DATA_BLOCK "CS_Drive_TL"   // DB14, Motion_DB
// stored: InstanceOfName TO_SynchronousAxis, OfSystemLibElement TO_SynchronousAxis, OfSystemLibVersion 7.0
TO_SynchronousAxis   // technology object, version 7.0
// stored: Connection Interface Actor, InputAddress 816, OutputAddress 816
// stored: Connection Interface Sensor[1], InputAddress 816, OutputAddress 816, SensorIndexInActorTelegram 1
   // // inherited from TO_PositioningAxis
   // // inherited from TO_SpeedAxis
   // // inherited from TO_Axis
   // // inherited from TO_Object
   // VAR
   //    Actor : TO_Struct_Actor;
   // END_VAR
   // VAR
   //    Sensor : Array[1..4] of TO_Struct_Sensor;
   //    PositionControl : TO_Struct_PositionControl;
   // END_VAR
   // VAR
   //    StatusSynchronizedMotion { ExternalWritable := 'False'; S7_SetPoint := 'True'} : TO_Struct_StatusSynchronizedMotion;
   // END_VAR
BEGIN
   Actor.Interface.AddressIn.RID := 16#208072a;
   Actor.Interface.AddressIn.AREA := 16#81;
   Actor.Interface.AddressIn.OFFSET := 816;
   Actor.Interface.AddressOut.RID := 16#208072b;
   Actor.Interface.AddressOut.AREA := 16#82;
   Actor.Interface.AddressOut.OFFSET := 816;
   Sensor[1].Interface.AddressIn.RID := 16#208072a;
   Sensor[1].Interface.AddressIn.AREA := 16#81;
   Sensor[1].Interface.AddressIn.OFFSET := 816;
   Sensor[1].Interface.AddressOut.RID := 16#208072b;
   Sensor[1].Interface.AddressOut.AREA := 16#82;
   Sensor[1].Interface.AddressOut.OFFSET := 816;
   PositionControl.EnableDSC := true;
   _Actor.Interface.Telegram := 105;
   _Sensor[1].Interface.Telegram := 105;
END_DATA_BLOCK

DATA_BLOCK "CS_Drive_TP"   // DB13, Motion_DB
// stored: InstanceOfName TO_SynchronousAxis, OfSystemLibElement TO_SynchronousAxis, OfSystemLibVersion 7.0
TO_SynchronousAxis   // technology object, version 7.0
// stored: Connection Interface Actor, InputAddress 608, OutputAddress 608
// stored: Connection Interface Sensor[1], InputAddress 608, OutputAddress 608, SensorIndexInActorTelegram 1
   // // inherited from TO_PositioningAxis
   // // inherited from TO_SpeedAxis
   // // inherited from TO_Axis
   // // inherited from TO_Object
   // VAR
   //    Actor : TO_Struct_Actor;
   // END_VAR
   // VAR
   //    Sensor : Array[1..4] of TO_Struct_Sensor;
   //    PositionControl : TO_Struct_PositionControl;
   // END_VAR
   // VAR
   //    StatusSynchronizedMotion { ExternalWritable := 'False'; S7_SetPoint := 'True'} : TO_Struct_StatusSynchronizedMotion;
   // END_VAR
BEGIN
   Actor.Interface.AddressIn.RID := 16#208072a;
   Actor.Interface.AddressIn.AREA := 16#81;
   Actor.Interface.AddressIn.OFFSET := 608;
   Actor.Interface.AddressOut.RID := 16#208072b;
   Actor.Interface.AddressOut.AREA := 16#82;
   Actor.Interface.AddressOut.OFFSET := 608;
   Sensor[1].Interface.AddressIn.RID := 16#208072a;
   Sensor[1].Interface.AddressIn.AREA := 16#81;
   Sensor[1].Interface.AddressIn.OFFSET := 608;
   Sensor[1].Interface.AddressOut.RID := 16#208072b;
   Sensor[1].Interface.AddressOut.AREA := 16#82;
   Sensor[1].Interface.AddressOut.OFFSET := 608;
   PositionControl.EnableDSC := true;
   _Actor.Interface.Telegram := 105;
   _Sensor[1].Interface.Telegram := 105;
END_DATA_BLOCK

DATA_BLOCK "CS_Virtual_Axis"   // DB22, Motion_DB
// stored: InstanceOfName TO_PositioningAxis, OfSystemLibElement TO_PositioningAxis, OfSystemLibVersion 7.0
TO_PositioningAxis   // technology object, version 7.0
   // // inherited from TO_SpeedAxis
   // // inherited from TO_Axis
   // // inherited from TO_Object
   // VAR
   //    VirtualAxis : TO_Struct_VirtualAxis;
   // END_VAR
   // VAR
   //    Position { ExternalWritable := 'False'} : LReal;
   //    ActualPosition { ExternalWritable := 'False'} : LReal;
   //    ActualVelocity { ExternalWritable := 'False'} : LReal;
   //    ActualAcceleration { ExternalWritable := 'False'} : LReal;
   //    OperativeSensor { ExternalWritable := 'False'} : UDInt;
   //    ModuloCycle { ExternalWritable := 'False'} : DInt;
   //    ActualModuloCycle { ExternalWritable := 'False'} : DInt;
   //    Clamping { S7_SetPoint := 'True'} : TO_Struct_Clamping;
   //    Sensor { S7_SetPoint := 'True'} : Array[1..4] of TO_Struct_Sensor;
   //    Extrapolation { S7_SetPoint := 'True'} : TO_Struct_Extrapolation;
   //    Mechanics { S7_SetPoint := 'True'} : TO_Struct_Mechanics;
   //    Properties { ExternalWritable := 'False'; S7_SetPoint := 'True'} : TO_Struct_Properties;
   //    Modulo { S7_SetPoint := 'True'} : TO_Struct_Modulo;
   //    PositionLimits_SW { S7_SetPoint := 'True'} : TO_Struct_PositionLimitsSW;
   //    PositionLimits_HW { S7_SetPoint := 'True'} : TO_Struct_PositionLimitsHW;
   //    Homing { S7_SetPoint := 'True'} : TO_Struct_Homing;
   //    PositionControl { S7_SetPoint := 'True'} : TO_Struct_PositionControl;
   //    SetpointFilter { S7_SetPoint := 'True'} : TO_Struct_SetpointFilter;
   //    DynamicAxisModel { S7_SetPoint := 'True'} : TO_Struct_DynamicAxisModel;
   //    FollowingError { S7_SetPoint := 'True'} : TO_Struct_FollowingError;
   //    CrossPlcSynchronousOperation { S7_SetPoint := 'True'} : TO_Struct_CrossPlcSynchronousOperation;
   //    PositioningMonitoring { S7_SetPoint := 'True'} : TO_Struct_PositioningMonitoring;
   //    StandstillSignal { S7_SetPoint := 'True'} : TO_Struct_StandstillSignal;
   //    StatusPositioning { ExternalWritable := 'False'; S7_SetPoint := 'True'} : TO_Struct_StatusPositioning;
   //    StatusServo { ExternalWritable := 'False'; S7_SetPoint := 'True'} : TO_Struct_StatusServo;
   //    StatusProvidedLeadingValue { ExternalWritable := 'False'; S7_SetPoint := 'True'} : TO_Struct_StatusProvidedLeadingValue;
   //    StatusSensor { ExternalWritable := 'False'; S7_SetPoint := 'True'} : Array[1..4] of TO_Struct_StatusSensor;
   //    StatusExtrapolation { ExternalWritable := 'False'; S7_SetPoint := 'True'} : TO_Struct_StatusExtrapolation;
   //    StatusKinematicsMotion { ExternalWritable := 'False'; S7_SetPoint := 'True'} : TO_Struct_StatusKinematicsMotion;
   // END_VAR
BEGIN
   VirtualAxis.Mode := 1;
   FollowingError.WarningLevel := 64.0;
   VirtualAxis.Mode := 1;
END_DATA_BLOCK
